// TIA Portal V17 export
// export: Created 2024-09-02T12:50:30.0462005Z, ExportSetting WithDefaults, DisplayName Totally Integrated Automation Portal, DisplayVersion V17, DisplayName TIA Portal Openness, DisplayVersion V17, DisplayName TIA Portal Version Control Interface, DisplayVersion V17, DisplayName STEP 7 Professional, DisplayVersion V17, DisplayName STEP 7 Safety, DisplayVersion V17, DisplayName WinCC Professional, DisplayVersion V17
TYPE "a_MGBN"
// stored: IsFailsafeCompliant false
   STRUCT
      LEDNotHalt : Bool;   // Notausmodul - LED Not-Halt (optional) / Emergency stop module - LED emergency stop (optional)
      "res2.1" : Bool;   // Notausmodul - Reserve / Emergency stop module - reserve
      "res2.2" : Bool;   // Notausmodul - Reserve / Emergency stop module - reserve
      "res2.3" : Bool;   // Notausmodul - Reserve / Emergency stop module - reserve
      "res2.4" : Bool;   // Notausmodul - Reserve / Emergency stop module - reserve
      "res2.5" : Bool;   // Notausmodul - Reserve / Emergency stop module - reserve
      "res2.6" : Bool;   // Notausmodul - Reserve / Emergency stop module - reserve
      "res2.7" : Bool;   // Notausmodul - Reserve / Emergency stop module - reserve
      TürÖffnen : Bool;   // Zuhaltemodul - Magnet (Tür öffnen) / Blocking module - Magnet (open door)
      "res3.1" : Bool;   // Zuhaltemodul - Reserve / Blocking module - reserve
      "res3.2" : Bool;   // Zuhaltemodul - Reserve / Blocking module - reserve
      "res3.3" : Bool;   // Zuhaltemodul - Reserve / Blocking module - reserve
      "res3.4" : Bool;   // Zuhaltemodul - Reserve / Blocking module - reserve
      "res3.5" : Bool;   // Zuhaltemodul - Reserve / Blocking module - reserve
      "res3.6" : Bool;   // Zuhaltemodul - Reserve / Blocking module - reserve
      "res3.7" : Bool;   // Zuhaltemodul - Reserve / Blocking module - reserve
      Quittierung : Bool;   // Diagnose - Quittierung / Diagnosis - Acknowledgement
      Reset : Bool;   // Diagnose - Reset MGB / Diagnosis - Reset MGB
      "res4.2" : Bool;   // Diagnose - Reserve / Diagnosis - Reserve
      "res4.3" : Bool;   // Diagnose - Reserve / Diagnosis - Reserve
      "res4.4" : Bool;   // Diagnose - Reserve / Diagnosis - Reserve
      "res4.5" : Bool;   // Diagnose - Reserve / Diagnosis - Reserve
      "res4.6" : Bool;   // Diagnose - Reserve / Diagnosis - Reserve
      "res4.7" : Bool;   // Diagnose - Reserve / Diagnosis - Reserve
   END_STRUCT;
END_TYPE
